# B&R Automation Studio project AutomationStudio_lab1
Automation Studio 4.5.2.102

## Configuration Config1

### Hardware
```
4PP065_0571_P74 : 4PP065.0571-P74 v1.1.2.0
  Connector IF5:
    ActivateDevice = 1
    Mode = Manual
    InternetAddress = 10.0.1.10
    SubnetMask = 255.255.255.0
  ConfigurationID = lab1_Config1
  Simulation = 1
```

## Logical view

### Library Logical/Libraries/Library

#### Library.fun
```iecst
{REDUND_ERROR} FUNCTION_BLOCK FB_Integrator (*TODO: Add your comment here*) (*$GROUP=User,$CAT=User,$GROUPICON=User.png,$CATICON=User.png*)
	VAR_INPUT
		in : {REDUND_UNREPLICABLE} REAL;
	END_VAR
	VAR_OUTPUT
		out : REAL;
	END_VAR
	VAR
		dt : REAL;
		prev_value : REAL;
	END_VAR
END_FUNCTION_BLOCK

{REDUND_ERROR} FUNCTION_BLOCK FB_Motor (*TODO: Add your comment here*) (*$GROUP=User,$CAT=User,$GROUPICON=User.png,$CATICON=User.png*)
	VAR_INPUT
		u : REAL;
	END_VAR
	VAR_OUTPUT
		w : REAL;
		phi : REAL;
	END_VAR
	VAR
		integrator1 : FB_Integrator;
		integrator2 : FB_Integrator;
		Tm : REAL;
		ke : REAL;
		dt : REAL;
	END_VAR
END_FUNCTION_BLOCK

{REDUND_ERROR} FUNCTION_BLOCK FB_Regulator (*TODO: Add your comment here*) (*$GROUP=User,$CAT=User,$GROUPICON=User.png,$CATICON=User.png*)
	VAR_INPUT
		e : REAL;
	END_VAR
	VAR_OUTPUT
		u : REAL;
	END_VAR
	VAR
		k_p : REAL;
		k_i : REAL;
		integrator : FB_Integrator;
		iyOld : REAL;
		max_abs_value : REAL;
		dt : REAL;
		temp : REAL;
		temp_pos : REAL;
		temp2 : REAL;
	END_VAR
END_FUNCTION_BLOCK
```

#### FB_Integrator.c
```c
#include <bur/plctypes.h>
#ifdef __cplusplus
	extern "C"
	{
#endif
	#include "Library.h"
#ifdef __cplusplus
	};
#endif
/* TODO: Add your comment here */
void FB_Integrator(struct FB_Integrator* inst)
{
	inst->out = inst->dt * inst->in + inst->prev_value;
	inst->prev_value = inst->out;
}
```

#### FB_Motor.c
```c
#include <bur/plctypes.h>
#ifdef __cplusplus
	extern "C"
	{
#endif
	#include "Library.h"
#ifdef __cplusplus
	};
#endif
/* TODO: Add your comment here */
void FB_Motor(struct FB_Motor* inst)
{

	inst->integrator1.dt = inst->dt/inst->Tm;
	inst->integrator2.dt = inst->dt;

	inst->integrator1.in = inst->u / inst->ke - inst->w;
	FB_Integrator(&inst->integrator1);
	inst->integrator2.in = inst->integrator1.out;
	FB_Integrator(&inst->integrator2);
	inst->w = inst->integrator1.out;
	inst->phi = inst->integrator2.out;
}
```

#### FB_Regulator.c
```c
#include <bur/plctypes.h>
#ifdef __cplusplus
	extern "C"
	{
#endif
	#include "Library.h"
#ifdef __cplusplus
	};
#endif
/* TODO: Add your comment here */
void FB_Regulator(struct FB_Regulator* inst)
{

	inst->integrator.dt = inst->dt;

	inst->temp = inst->e * inst->k_p > inst->max_abs_value ? inst->max_abs_value : inst->e * inst->k_p;
	inst->temp = inst->e * inst->k_p < -inst->max_abs_value ? -inst->max_abs_value : inst->e * inst->k_p;

	inst->integrator.in = inst->e * inst->k_i + inst->temp_pos;
	FB_Integrator(&inst->integrator);

	inst->temp += inst->integrator.out;
	inst->temp2 = inst->temp;

	inst->temp = inst->temp > inst->max_abs_value ? inst->max_abs_value : inst->temp;
	inst->temp = inst->temp < -inst->max_abs_value ? -inst->max_abs_value : inst->temp;

	inst->temp_pos = inst->temp - inst->temp2;

	inst->u = inst->temp;
}
```

### Program Logical/Program

#### Variables.var
```iecst
VAR
	fb_controller_1 : FB_Regulator;
	fb_controller_2 : FB_Regulator;
	fb_controller : FB_Regulator;
	fb_motor : FB_Motor;
	Speed : REAL := 10;
	Enable : BOOL := FALSE;
	feedback_1 : REAL;
	feedback_2 : REAL;
	feedback : REAL;
	feedback_without_con : REAL;
	counter : USINT;
	fb_motor_1 : FB_Motor;
	fb_motor_2 : FB_Motor;
	fb_motor_without_con : FB_Motor;
END_VAR
```

#### Cyclic.c
```c
#include <bur/plctypes.h>

#ifdef _DEFAULT_INCLUDES
	#include <AsDefault.h>
#endif

void _CYCLIC ProgramCyclic(void)
{
	fb_motor.ke = 0.24;
	fb_motor.Tm = 0.1;
	fb_motor.dt = 0.1;

	fb_motor_without_con.ke = 0.24;
	fb_motor_without_con.Tm = 0.1;
	fb_motor_without_con.dt = 0.1;

	fb_controller.k_i = 7.2;
	fb_controller.k_p = 0.78;
	fb_controller.max_abs_value = 24;
	fb_controller.temp_pos = 0;
	fb_controller.dt = 0.1;

	fb_motor_1.ke = 0.0241;
	fb_motor_1.Tm = 0.0226;
	fb_motor_1.dt = 0.01;

	fb_controller_1.k_i = 0.8;
	fb_controller_1.k_p = 0.018;
	fb_controller_1.max_abs_value = 24;
	fb_controller_1.temp_pos = 0;
	fb_controller_1.dt = 0.01;

	fb_motor_2.ke = 0.0735;
	fb_motor_2.Tm = 0.0147;
	fb_motor_2.dt = 0.01;

	fb_controller_2.k_i = 2.45;
	fb_controller_2.k_p = 0.036;
	fb_controller_2.max_abs_value = 24;
	fb_controller_2.temp_pos = 0;
	fb_controller_2.dt = 0.01;

	if(counter == 200)
	{
		Speed = 0;
		counter = 0;
	}
	if (counter == 50)
	{
		Speed = 50;
	}
	counter++;
	if (Enable)
	{
		fb_motor_without_con.u = Speed - feedback_without_con;
		FB_Motor(&fb_motor_without_con);

		feedback_without_con = fb_motor_without_con.w;

		fb_controller.e = Speed - feedback;
		FB_Regulator(&fb_controller);

		fb_motor.u = fb_controller.u;
		FB_Motor(&fb_motor);

		feedback = fb_motor.w;

		fb_controller_1.e = Speed - feedback_1;
		FB_Regulator(&fb_controller_1);

		fb_motor_1.u = fb_controller_1.u;
		FB_Motor(&fb_motor_1);

		feedback_1 = fb_motor_1.w;

		fb_controller_2.e = Speed - feedback_2;
		FB_Regulator(&fb_controller_2);

		fb_motor_2.u = fb_controller_2.u;
		FB_Motor(&fb_motor_2);

		feedback_2 = fb_motor_2.w;
	}

}
```

#### Init.c
```c
#include <bur/plctypes.h>

#ifdef _DEFAULT_INCLUDES
	#include <AsDefault.h>
#endif

void _INIT ProgramInit(void)
{
	Speed = 0;
	counter = 0;
}
```
